TEXTLIST EventScheme
  0 = '0 - Instance type and number'
  1 = '1 - Short address and instance type'
  2 = '2 - Short address and instance number'
  3 = '3 - Device group and instance type'
  4 = '4 - Instance group and instance type'
   = ''
END_TEXTLIST

(* stored: Version 1.1.0.1, ProductVersion 3.1.4024.9
   TextList EventScheme: Id {416ddd96-e463-443c-a16e-b4eaace0f971} *)
